// TwinCAT 3 PLC project PLC1
// ProgramVersion: 3.1.4024.0
// libraries:
//   Tc2_ControllerToolbox, * (Beckhoff Automation GmbH)
//   Tc2_MC2, * (Beckhoff Automation GmbH)
//   Tc2_Standard, * (Beckhoff Automation GmbH)
//   Tc2_System, * (Beckhoff Automation GmbH)
//   Tc2_Utilities, * (Beckhoff Automation GmbH)
//   Tc3_Module, * (Beckhoff Automation GmbH)
//   Tc3_Vision, * (Beckhoff Automation GmbH)
// project tree:
//   DUTs/Motion/ E_MotionStates.TcDUT
//   DUTs/Vision/ E_Shapes.TcDUT
//   GVLs/ IO.TcGVL, Motion.TcGVL, Safety.TcGVL
//   / PlcTask.TcTTO
//   POUs/FIle IO/Reading/ FB_ReadReferenceShapeXMLFiles.TcPOU
//   POUs/Indicators/ FB_Flash.TcPOU
//   POUs/ MAIN.TcPOU
//   POUs/Motion/ PositionStateMachine.TcPOU
//   POUs/Vision/ BasicVision.TcPOU
// real-time tasks:
//   TASK PlcTask: cycle T#10ms, priority 20, ADS port 350
//   TASK VnTask ImgAcq (Camera1): cycle T#1ms, priority 5, ADS port 351
//   TASK VnTask ADS (Camera1): cycle T#10ms, priority 6, ADS port 352
// motion (NC):
//   TASK NC-Task 1 SAF: cycle T#2ms, priority 4, ADS port 501
//   TASK NC-Task 1 SVB: cycle T#10ms, priority 8, ADS port 511
//   AXIS Linear Slide (id 3)
//     Dynamic: Acceleration=5485.83, Deceleration=5485.83, Jerk=164575
//     Velo: RefSearch=3.65722, RefSync=3.65722, SlowManual=18.2861, FastManual=109.7166, Fast=365.722, Maximum=365.722
//     OtherSettings: AllowMotionCmdToSlave=true
//     encoder EncType=19
//       EncPara: ScaleFactorNumerator=4.064, ScaleFactorDenominator=1048576, MaxCount=#xffffffff
//         SoftEndMinControl: Range=-5
//         SoftEndMaxControl: Range=275
//     drive DrvType=16
//       DrvPara: MaxCount=#xffffffff, DriveControlDWord=#x00020100
//         Analog: VeloReferenz=402.2942, VeloScale=32, TorqueSetpointScale=10, ScaleFactorActTorque=0.1
//         TimeComp: TaskDelayCycles=1
//     controller CtrType=1
//       CtrPara: PriorControlFactor=1
//         PosDiffControl: Enable=false
//         Observer: BandWidth=20
// I/O:
//   DEVICE EK1100, AmsNetId 169.254.119.130.3.1
//     Term 2 (EK1100) [EK1100 EtherCAT Coupler (2A E-Bus)]
//       Term 3 (EL1012) [EL1012 2Ch. Dig. Input 24V, 10µs]
//       Term 4 (EL1252) [EL1252 2Ch. Fast Dig. Input 24V, 1µs, DC Latch]
//       Term 5 (EL1034) [EL1034 4Ch. Dig. Input 24V, potential-free, 10µs]
//       Term 6 (EL2024) [EL2024 4Ch. Dig. Output 24V, 2A]
//       Term 7 (ELM7222-9016) [ELM7222-9016 2Ch. Servo Terminal (48 V, 8 A RMS, OCT, STO, TwinSAFE Logic)]
//         modules: Module 1 (SAFETY)
//         startup 32785:21 := 0E01 // DRV Motor Settings Ch.1 / Commutation offset
//         startup 32785:27 := 10270000 // DRV Motor Settings Ch.1 / Motor speed limitation
//         startup 28688:11 := FC0D // DRV Outputs Ch.1 / Torque limitation
//         startup 32784:19 := FD00 // DRV Amplifier Settings Ch.1 / Current loop proportional gain
//         startup 32784:18 := 0600 // DRV Amplifier Settings Ch.1 / Current loop integral time
//         startup 32784:21 := 2B000000 // DRV Amplifier Settings Ch.1 / Velocity loop proportional gain
//         startup 32784:20 := 96000000 // DRV Amplifier Settings Ch.1 / Velocity loop integral time
//       Term 8 (EL1904) [EL1904, 4 Ch. Safety Input 24V, TwinSAFE]
//         modules: Module 1 (FSOES)
//       Term 16 (EL2004) [EL2004 4Ch. Dig. Output 24V, 0.5A]
//       Term 17 (EL9011) [EL9011 End Terminal]
//   DEVICE Device 1 (RT-Ethernet Adapter)
// variable links:
//   EK1100 <-> EK1100/Term 2 (EK1100)/Term 7 (ELM7222-9016)
//     Term 2 (EK1100)/Term 8 (EL1904)/Module 1 (FSOES)/TxPDO/FSOE <-> Module 1 (SAFETY)/SAFETY FSoE Connection 1 Receive Message/Message_4
//   EK1100 <-> EK1100/Term 2 (EK1100)/Term 8 (EL1904)
//     Term 2 (EK1100)/Term 7 (ELM7222-9016)/Module 1 (SAFETY)/SAFETY FSoE Connection 1 Send Message/Message_4 <-> Module 1 (FSOES)/RxPDO/FSOE
//   NC-Task 1 SAF/Axes/Linear Slide <-> EK1100/Term 2 (EK1100)/Term 7 (ELM7222-9016)
//     Drive/Inputs/In/nDataIn1 <-> DRV Following error actual value Channel 1/Following error actual value
//     Drive/Inputs/In/nDcOutputTime <-> InfoData/DcOutputShift
//     Drive/Inputs/In/nState1 <-> DRV Statusword Channel 1/Statusword
//     Drive/Inputs/In/nState2 <-> DRV Statusword Channel 1/Statusword @bit 8
//     Drive/Inputs/In/nState4 @bit 1 <-> WcState/InputToggle0
//     Drive/Inputs/In/nState4 <-> WcState/WcState0
//     Drive/Outputs/Out/nCtrl1 <-> DRV Controlword Channel 1/Controlword
//     Drive/Outputs/Out/nCtrl2 <-> DRV Controlword Channel 1/Controlword @bit 8
//     Drive/Outputs/Out/nDataOut1 <-> DRV Target position Channel 1/Target position
//     Enc/Inputs/In/nDataIn1 <-> FB Position Channel 1/Position
//     Enc/Inputs/In/nDcInputTime <-> InfoData/DcInputShift
//     Enc/Inputs/In/nState4 @bit 1 <-> WcState/InputToggle0
//     Enc/Inputs/In/nState4 <-> WcState/WcState0
//   PLC1/PLC1 Instance <-> EK1100/Term 2 (EK1100)/Term 16 (EL2004)
//     PlcTask Outputs/PositionStateMachine.bHandClosed <-> Channel 1/Output
//   PLC1/PLC1 Instance <-> EK1100/Term 2 (EK1100)/Term 3 (EL1012)
//     PlcTask Inputs/IO.bInSafetyRunSwitch <-> Channel 1/Input
//     PlcTask Inputs/PositionStateMachine.bRecalibrate <-> Channel 2/Input
//   PLC1/PLC1 Instance <-> EK1100/Term 2 (EK1100)/Term 4 (EL1252)
//     PlcTask Inputs/IO.bInAckSignal <-> Channel 1/Input
//   PLC1/PLC1 Instance <-> EK1100/Term 2 (EK1100)/Term 5 (EL1034)
//     PlcTask Inputs/PositionStateMachine.bLimitSwitch <-> Channel 1/Input
//   PLC1/PLC1 Instance <-> EK1100/Term 2 (EK1100)/Term 6 (EL2024)
//     PlcTask Outputs/MAIN.bLimitSwitchPower <-> Channel 2/Output
//     PlcTask Outputs/MAIN.bRingLight <-> Channel 1/Output
//   PLC1/PLC1 Instance <-> EK1100/Term 2 (EK1100)/Term 7 (ELM7222-9016)
//     PlcTask Outputs/Safety.bErrorAck <-> Module 1 (SAFETY)/SAFETY Standard Outputdata/Standard In Var 1
//     PlcTask Outputs/Safety.bSafetyRestart <-> Module 1 (SAFETY)/SAFETY Standard Outputdata/Standard In Var 7
//     PlcTask Outputs/Safety.bSafetyRun <-> Module 1 (SAFETY)/SAFETY Standard Outputdata/Standard In Var 2
//   PLC1/PLC1 Instance <-> NC-Task 1 SAF/Axes/Linear Slide
//     PlcTask Inputs/Motion.Servo.NcToPlc <-> Outputs/ToPlc
//     PlcTask Outputs/Motion.Servo.PlcToNc <-> Inputs/FromPlc

CONFIGURATION PLC1
    RESOURCE PLC ON TwinCAT3
        TASK PlcTask(INTERVAL := T#10ms, PRIORITY := 20);
        PROGRAM MAIN WITH PlcTask : MAIN;
    END_RESOURCE
END_CONFIGURATION

// ---- DUTs/Motion/E_MotionStates.TcDUT
//{attribute 'qualified_only'}
{attribute 'strict'}
TYPE E_MotionStates :
(
	// Initialize Motor
	eInitialize := 0,
	
	// Activate Calibration
	eActivateCalibration := 1,
	
	// Calibrate Position
	eCalibrate := 2,
	
	// Scan for shape
	eScanAndGrab := 3,
	
	// Open Hand
	eOpenHand := 4,
	
	// Close Hand
	eCloseHand := 5,
	
	// Position 10 : Start
	eSetTargetPosition_1 := 10,
	eRunToPosition_1 := 11,
	
	// Position 20 : Triangle Box
	eSetTargetPosition_2 := 20,
	eRunToPosition_2 := 21,
	
	// Position 30 : Square Box
	eSetTargetPosition_3 := 30,
	eRunToPosition_3 := 31,
	
	// Position 40 : Circle Box
	eSetTargetPosition_4 := 40,
	eRunToPosition_4 := 41,
	
	// Error Handling
	eErrorState1 := 999
);
END_TYPE

// ---- DUTs/Vision/E_Shapes.TcDUT
//{attribute 'qualified_only'}
{attribute 'strict'}
TYPE E_Shapes :
(
	// No shape
	eNoShape := -1,	

	// Triangle
	eTriangle := 0,
	
	// Circle
	eCircle := 1,
	
	// Square
	eSquare := 2
);
END_TYPE

// ---- GVLs/IO.TcGVL
{attribute 'qualified_only'}
VAR_GLOBAL
	// Acknowledge Error Button | Linked to GPB1
	bInAckSignal AT %I* : BOOL;
	// Safe to run Switch | Linked to GSS1
	bInSafetyRunSwitch AT %I* : BOOL;
	
	// Signal from TwinSAFE Controller | Linked to EStopIndicator Alias
	bInEStopSignal AT %I* : BOOL;
	// Light up indicator | Linked to RPBL1
	bOutEStopIndicator AT %Q* : BOOL;
END_VAR

// ---- GVLs/Motion.TcGVL
{attribute 'qualified_only'}
VAR_GLOBAL
	Servo : AXIS_REF;
END_VAR

// ---- GVLs/Safety.TcGVL
{attribute 'qualified_only'}
VAR_GLOBAL
	// PLC Outputs sent to TwinSAFE Controller
	bErrorAck AT %Q* : BOOL;
	bSafetyRun AT %Q* : BOOL;
	bSafetyRestart AT %Q* : BOOL;
END_VAR

// ---- POUs/MAIN.TcPOU
PROGRAM MAIN
VAR
	// ------------------------------------------- //
	// Outputs
	bLight_GPBL1 AT %Q* 	: 	BOOL;
	bLight_GSSL1 AT %Q* 	: 	BOOL;
	
	// ------------------------------------------- //
	// Motion
	bLimitSwitchPower AT %Q*:	BOOL := TRUE;
	
	// ------------------------------------------- //
	// Indicators
	fbBlink : FB_Flash;
	
	// -------------------------------------------------------------------------------------- //
	// Vision
	bRingLight AT %Q*		:	BOOL := TRUE;
	hr						:	HRESULT;
	fbCamera 				:	FB_VN_GevCameraControl;
	eState 					: 	EtcVNCameraState;
	
	// Raw Input
	ipImageIn 				: 	ITcVnImage;
	
	// ------------------------------------------- //
	// Colors
	
	// Colored output to perform processing on
	ipImageWork 			: 	ITcVnImage;
	ipImageWorkDisp 		: 	ITcVnDisplayableImage;
	
	// Color maps to black and white output
	// ** Could also check for ranges [0,0,0] to [199,255,255] to go straight to proper color map **
	ipImageColorMap_White 	: 	ITcVnImage;
	aColorLow_White 		: 	TcVnVector4_LREAL := [199,255,255];
	aColorHigh_White 		: 	TcVnVector4_LREAL := [255,255,255];
	
	// Invert image so that objects are white and background is black
	ipImageColorMap_Black	: 	ITcVnImage;
	ipImageColorMapDisp_Black : ITcVnDisplayableImage;
	
	// Processed Output
	ipImageResult 			:	ITcVnImage;
	ipImageResultDisp 		: 	ITcVnDisplayableImage;
	
	
	// ------------------------------------------- //
	// Contours
	
	ipContourList 			: 	ITcVnContainer;				// Container of containers containing points for contours
	ipContourListIterator	: 	ITcVnForwardIterator;		// Used to dynamically iterate through ContourList
	ipContour				: 	ITcVnContainer;				// A single contour
	
	aColor_Green			: 	TcVnVector4_LREAL := [0,255,0]; // Constant value, color of drawn contours
	
	// ------------------------------------------- //
	// Object Detection
	
	// Load Reference FIles
	bFilesRead				: 	BOOL := FALSE;
	fbReadReferenceShapeFiles : FB_ReadReferenceShapeXMLFiles;
		
	ipReference_Triangle	: 	ITcVnContainer;				// Destination container for our triangle	
	ipReference_Circle		: 	ITcVnContainer;				// Destination container for our circle
	ipReference_Square		: 	ITcVnContainer;				// Destination container for our square																		
	
	// Calculate area and dissimilarity to determine correct shape type
	fArea					: 	LREAL;						// Area of found contours
	
	fTriangleDissimilarity	: 	LREAL;						// Dissimilarity between reference triangle and actual images
	fCircleDissimilarity	: 	LREAL;						// Dissimilarity between reference circle and actual images
	fSquareDissimilarity	: 	LREAL;						// Dissimilarity between reference square and actual images
	fMinimumDissimilarity	: 	LREAL;						
	
	sText					:	STRING(256);				// Text label on contour
	aCenter					:	TcVnPoint2_LREAL;			// Center of mass of contour
	
	iShape					: 	E_SHAPES := -1;				// Detected shape to be sent to PositionStateMachine
END_VAR

_AppInfo.KeepOutputsOnBP := TRUE;

// Safety Handling
Safety.bSafetyRestart := IO.bInAckSignal;
Safety.bErrorAck := IO.bInAckSignal;
Safety.bSafetyRun := IO.bInSafetyRunSwitch; // ** HARDWIRED TO TRUE **

// Indicators
bLight_GPBL1 := IO.bInAckSignal;
bLight_GSSL1 := IO.bInSafetyRunSwitch;

fbBlink(bEnable:= NOT IO.bInEStopSignal, tTimeOn:= T#500MS, tTimeOff:= T#500MS, bPulse=> IO.bOutEStopIndicator);

// -------------------------------------------------------------------------------------- //
// Vision
	
// Read in reference image files
IF NOT bFilesRead THEN
	fbReadReferenceShapeFiles(
		ipReference_Triangle => ipReference_Triangle,
		ipReference_Circle => ipReference_Circle,
		ipReference_Square => ipReference_Square
	);
	
	bFilesRead := fbReadReferenceShapeFiles.bAllFilesLoaded;
END_IF

IF bFilesRead THEN
	eState := fbCamera.GetState();
	hr := S_OK;
		
	IF eState <= TCVN_CS_ERROR THEN // If state is in error, attempt reset
		hr := fbCamera.Reset();
	ELSIF eState < TCVN_CS_ACQUIRING THEN
		hr := fbCamera.StartAcquisition();
	ELSIF eState = TCVN_CS_ACQUIRING THEN
		// Get current image and set ROI
		hr := fbCamera.GetCurrentImage(ipImageIn);
		//hr := F_VN_SetRoi(953, 480, 450, 370, ipImageIn, hr); 
			
		// Check if image was successfully recieved
		IF SUCCEEDED(hr) AND ipImageIn <> 0 THEN
			// Color Detection
		
			// Create working colored image and displayable version
			hr := F_VN_ConvertColorSpace(ipImageIn, ipImageWork,TCVN_CST_BAYER_RG_TO_RGB, hr);
			hr := F_VN_CopyIntoDisplayableImage(ipImageWork, ipImageWorkDisp, hr);
			
			// Copy our work image into final image for later use during contour drawing
			hr := F_VN_CopyImage(ipImageWork, ipImageResult, hr);
			
			// Increase contrast by converting anything that isn't pure white to black
			// This creates a white image with black shapes on it
			hr := F_VN_CheckColorRange(ipImageWork, ipImageColorMap_White, aColorLow_White, aColorHigh_White, hr);
			
			// Invert white color map to a black color map 
			// This creates a black image with white shapes on it
			hr := F_VN_InvertImageColor(ipImageColorMap_White, ipImageColorMap_Black, hr);
			hr := F_VN_CopyIntoDisplayableImage(ipImageColorMap_Black, ipImageColorMapDisp_Black,hr);
			
			// ------------------------------------------- //
			// Contours
			
			// Use color map to find contours
			hr := F_VN_FindContours(ipImageColorMap_Black, ipContourList,hr);
			
			
			// ** DELETE WHEN ALL REFERENCES CREATED **
			// Count the number of contours and store in iContourSize
			// Write points to XML file
			hr := F_VN_GetForwardIterator(ipContourList, ipContourListIterator, hr);
		
			// Evaluate each subcontainer for contour points
			WHILE SUCCEEDED(hr) AND_THEN ipContourListIterator.CheckIfEnd() <> S_OK DO
				hr := F_VN_GetContainer(ipContourListIterator, ipContour, hr);
				hr := F_VN_IncrementIterator(ipContourListIterator, hr);
				
				// Draw contours
				hr := F_VN_DrawContours(ipContour, -1, ipImageResult, aColor_Green, 3, hr);
				
				// ------------------------------------------- //
				// Shape Detection
				
				// Determine area of contours to save resources scanning miscellaneous junk
				hr := F_VN_ContourArea(ipContour, fArea, hr);
				
				// Compare contours to reference images and determine closest match
				IF fArea > 10000 THEN
					hr := F_VN_MatchContours(ipContour, ipReference_Triangle, TCVN_CMCM_CONTOURS_MATCH_I1, fTriangleDissimilarity, hr);
					
					IF fTriangleDissimilarity < 0.0006 THEN
						iShape := eCircle;
						sText := 'Circle';
					ELSIF fTriangleDissimilarity >= 0.028 AND fTriangleDissimilarity <= 0.033 THEN
						iShape := eSquare;
						sText := 'Square';
					ELSIF fTriangleDissimilarity >= 0.122 AND fTriangleDissimilarity <= 0.144 THEN
						iShape := eTriangle;
						sText := 'Triangle';
					ELSE
						iShape := eNoShape;
						sText := 'Unknown';
					END_IF
				END_IF
				
				// Calculate center of mass and place text onto shape
				hr := F_VN_ContourCenterOfMass(ipContour, aCenter, hr);
				hr := F_VN_PutText(sText, ipImageResult, LREAL_TO_UDINT(aCenter[0] - 60), LREAL_TO_UDINT(aCenter[1] + 10), ETcVnFontType.TCVN_FT_HERSHEY_PLAIN, 2, aColor_Green,hr);
			END_WHILE
			
			hr := F_VN_CopyIntoDisplayableImage(ipImageResult, ipImageResultDisp, hr);
			
		END_IF
	END_IF
	
	// Call to PositionStateMachine to run motion
	PositionStateMachine(iShape := iShape);
END_IF

END_PROGRAM

// ---- POUs/Indicators/FB_Flash.TcPOU
FUNCTION_BLOCK FB_Flash
VAR_INPUT
	bEnable : BOOL;
	tTimeOn : TIME;
	tTimeOff : TIME;
END_VAR
VAR_OUTPUT
	bPulse : BOOL;
END_VAR
VAR
	fbTON : TON; // Timer on delay function block
	fbTOF : TOF; // Timer off delay function block
END_VAR

fbTON(IN := bEnable AND NOT fbTOF.Q, PT := tTimeOff, Q => , ET => );
fbTOF(IN := fbTON.Q, PT := tTimeOn, Q => bPulse, ET => );

END_FUNCTION_BLOCK

// ---- POUs/FIle IO/Reading/FB_ReadReferenceShapeXMLFiles.TcPOU
FUNCTION_BLOCK FB_ReadReferenceShapeXMLFiles

VAR_INPUT
END_VAR

VAR_OUTPUT
	ipReference_Triangle	: 	ITcVnContainer;		// Destination container for our triangle	
	ipReference_Circle		: 	ITcVnContainer;		// Destination container for our circle
	ipReference_Square		: 	ITcVnContainer;		// Destination container for our square
	bAllFilesLoaded			:	BOOL := FALSE;		// Triangle, Circle, and Square files are all loaded
END_VAR

VAR
	fbReadContainer			: 	FB_VN_ReadContainer;// Reads container and compares it to reference
	
	bTriangleReferenceLoaded: 	BOOL := FALSE;		// Triangle file is loaded
	bCircleReferenceLoaded	: 	BOOL := FALSE;		// Circle file is loaded		
	bSquareReferenceLoaded	: 	BOOL := FALSE;		// Square file is loaded

	sTriangleFilePath		: 	STRING(256) := 'C:\Users\Administrator\Documents\Vision\Shapes\ContourTemplates\Original\triangle.xml';		// File path to reference triangle on target system
	sCircleFilePath			: 	STRING(256) := 'C:\Users\Administrator\Documents\Vision\Shapes\ContourTemplates\Original\circle.xml';		// File path to reference circle on target system
	sSquareFilePath			: 	STRING(256) := 'C:\Users\Administrator\Documents\Vision\Shapes\ContourTemplates\Original\rectangle.xml';	// File path to reference square on target system
	
	nTriangleReadId			: 	INT := 0;
	nCircleReadId			: 	INT := 0;
	nSquareReadId			: 	INT := 0;
END_VAR

// Read Triangle
IF NOT bTriangleReferenceLoaded THEN
	fbReadContainer(
		sFilePath:= sTriangleFilePath, 
		ipDestContainer:= ipReference_Triangle, 
		nDestTypeGuid:= , 
		bRead:= TRUE, 
		nTimeout:= T#5S, 
	);
	
	IF NOT fbReadContainer.bBusy THEN
		IF nTriangleReadId >= 2 THEN
			bTriangleReferenceLoaded := TRUE;
		ELSE
			nTriangleReadId := nTriangleReadId + 1;
			fbReadContainer(sFilePath := sTriangleFilePath, bRead := FALSE);
		END_IF
	END_IF
END_IF

// Read Circle
IF NOT bCircleReferenceLoaded THEN
	fbReadContainer(
		sFilePath:= sCircleFilePath, 
		ipDestContainer:= ipReference_Circle, 
		nDestTypeGuid:= , 
		bRead:= TRUE, 
		nTimeout:= T#5S, 
	);
	
	IF NOT fbReadContainer.bBusy THEN
		IF nCircleReadId >= 2 THEN
			bCircleReferenceLoaded := TRUE;
		ELSE
			nCircleReadId := nCircleReadId + 1;
			fbReadContainer(sFilePath := sCircleFilePath, bRead := FALSE);
		END_IF
	END_IF
END_IF

// Read Square
IF NOT bSquareReferenceLoaded THEN
	fbReadContainer(
		sFilePath:= sSquareFilePath, 
		ipDestContainer:= ipReference_Square, 
		nDestTypeGuid:= , 
		bRead:= TRUE, 
		nTimeout:= T#5S, 
	);
	
	IF NOT fbReadContainer.bBusy THEN
		IF nSquareReadId >= 2 THEN
			bSquareReferenceLoaded := TRUE;
		ELSE
			nSquareReadId := nSquareReadId + 1;
			fbReadContainer(sFilePath := sSquareFilePath, bRead := FALSE);
		END_IF
	END_IF
END_IF

IF bTriangleReferenceLoaded AND bSquareReferenceLoaded AND bCircleReferenceLoaded THEN
	bAllFilesLoaded := TRUE;
END_IF

END_FUNCTION_BLOCK

// ---- POUs/Motion/PositionStateMachine.TcPOU
PROGRAM PositionStateMachine
VAR_INPUT
	iShape 					: 	INT;
END_VAR
VAR
	// State Machine
	iMotionStep 			: 	E_MotionStates;
	iNextTargetPosition		:	E_MotionStates;
	iResetState				: 	INT;
	
	// Motion
	iRunSpeed 				: 	INT := 100;
	iTargetPosition			:	INT;
	bExecuteMotion			:	BOOL;
	bRecalibrate AT %I*		:	BOOL;
	iPosition AT %Q* 		: 	LREAL;
	
	fbMotorEnable 			: 	MC_Power;
	fbMoveAbsolute 			: 	MC_MoveAbsolute;
	fbMoveVelocity			:	MC_MoveVelocity;
	fbSetPosition			:	MC_SetPosition;
	fbMotorStop 			: 	MC_Stop;
	fbMotorReset 			: 	MC_Reset;
	fbReadPosition 			: 	MC_ReadActualPosition;
	
	bServoAxisError AT %I* 	: 	BOOL;
	
	bLimitSwitch AT %I*		:	BOOL;
	bHandClosed AT %Q*		:	BOOL;
	
	// Timers
	tHandActuationTimer		:	TON;
	tVisionPauseTimer		:	TON;
	bStartHandTimer			:	BOOL;
	bStartVisionTimer		:	BOOL;
	
	// Vision
	hr						:	HRESULT;
	iNumberOfContours		:	ULINT;
END_VAR

Motion.Servo.ReadStatus();
fbReadPosition(
	Axis:= Motion.Servo, 
	Enable:= TRUE,  
	Position=> iPosition
);

IF bRecalibrate AND NOT fbMoveAbsolute.Busy AND NOT fbMoveVelocity.Busy AND NOT Motion.Servo.Status.Moving AND NOT Motion.Servo.Status.Error THEN
	iMotionStep := eActivateCalibration;
END_IF

	
CASE iMotionStep OF
	
	eInitialize : // Axis Ready
	
		fbMotorEnable(
			Axis:= Motion.Servo, 
			Enable:= TRUE, 
			Enable_Positive:= TRUE, 
			Enable_Negative:= TRUE, 
		);
	
		IF fbMotorEnable.Status THEN
			iMotionStep := eActivateCalibration;
		END_IF
		
	// -------------------------------------------------- //
		
	eActivateCalibration : // Activate Calibration
		bHandClosed := FALSE;
		
		IF bLimitSwitch THEN // Switch is not pressed, calibrate
			fbMoveVelocity(
				Axis:= Motion.Servo, 
				Execute:= TRUE , 
				Velocity:= 20, 
				Direction:= MC_Negative_Direction, 
			);
			iMotionStep := eCalibrate;
		ELSE // Switch is pressed, do not calibrate
			fbMoveVelocity(Axis:= Motion.Servo, Execute:= FALSE);
			fbSetPosition(Axis:= Motion.Servo, Execute:= TRUE, Position:= 0);
			iMotionStep := eSetTargetPosition_1;
		END_IF
		
		IF fbMoveAbsolute.Error THEN
			iMotionStep := eErrorState1;
		END_IF
	
	// -------------------------------------------------- //
	
	eCalibrate : // Axis Calibrating
		fbMoveVelocity(
			Axis:= Motion.Servo, 
			Execute:= FALSE , 
		);
		
		IF NOT bLimitSwitch AND NOT fbMoveVelocity.Busy THEN
			fbSetPosition(Axis:= Motion.Servo, Execute:= TRUE, Position:= 0);
			iMotionStep := eSetTargetPosition_1;
		ELSIF fbMoveVelocity.Error THEN
			iMotionStep := eErrorState1;
		END_IF
	
	// -------------------------------------------------- //
	
	eSetTargetPosition_1 : // Target Position : Start (0mm)
		iTargetPosition := 0;
		bExecuteMotion := TRUE;
		IF fbMoveAbsolute.Busy THEN
			iMotionStep := eRunToPosition_1;
		END_IF
		
		IF fbMoveAbsolute.Error THEN
			iMotionStep := eErrorState1;
		END_IF
	
	// -------------------------------------------------- //
	
	eRunToPosition_1 : // Run to Target Position : Start
		bExecuteMotion := FALSE;
		
		IF fbMoveAbsolute.Done AND NOT fbMoveAbsolute.Busy THEN
			iMotionStep := eScanAndGrab;
		ELSIF fbMoveAbsolute.Error THEN
			iMotionStep := eErrorState1;
		END_IF
	
	// -------------------------------------------------- //
	
	eSetTargetPosition_2 : // Set Target Position : Triangle Box (90mm)
		iTargetPosition := 90;
		bExecuteMotion := TRUE;
		
		iMotionStep := eRunToPosition_2;
		
		IF fbMoveAbsolute.Error THEN
			iMotionStep := eErrorState1;
		END_IF
	
	// -------------------------------------------------- //
	
	eRunToPosition_2 : // Run to Target Position : Triangle Box
		bExecuteMotion := FALSE;
		IF fbMoveAbsolute.Done AND NOT fbMoveAbsolute.Busy THEN
			iMotionStep := eOpenHand;
		ELSIF fbMoveAbsolute.Error THEN
			iMotionStep := eErrorState1;
		END_IF
	
	// -------------------------------------------------- //
	
	eSetTargetPosition_3 : // Set Target Position : Square Box (180mm)
		iTargetPosition := 180;
		bExecuteMotion := TRUE;
		IF fbMoveAbsolute.Busy THEN
			iMotionStep := eRunToPosition_3;
		END_IF
		
		IF fbMoveAbsolute.Error THEN
			iMotionStep := eErrorState1;
		END_IF
	
	// -------------------------------------------------- //
	
	eRunToPosition_3 : // Run to Target Position : Square Box
		bExecuteMotion := FALSE;
		IF fbMoveAbsolute.Done AND NOT fbMoveAbsolute.Busy THEN
			iMotionStep := eOpenHand;
		ELSIF fbMoveAbsolute.Error THEN
			iMotionStep := eErrorState1;
		END_IF
	
	// -------------------------------------------------- //
	
	eSetTargetPosition_4 : // Set Target Position : Circle Box (270mm)
		iTargetPosition := 270;
		bExecuteMotion := TRUE;
		IF fbMoveAbsolute.Busy THEN
			iMotionStep := eRunToPosition_4;
		END_IF
		
		IF fbMoveAbsolute.Error THEN
			iMotionStep := eErrorState1;
		END_IF
	
	// -------------------------------------------------- //
	
	eRunToPosition_4 : // Run to Target Position : Circle Box
		bExecuteMotion := FALSE;
		
		IF fbMoveAbsolute.Done AND NOT fbMoveAbsolute.Busy THEN
			iMotionStep := eOpenHand;
		ELSIF fbMoveAbsolute.Error THEN
			iMotionStep := eErrorState1;
		END_IF
	
	// -------------------------------------------------- //
	
	eScanAndGrab : // Scan for shape and Grab
		hr := F_VN_GetNumberOfElements(Main.ipContourList, iNumberOfContours, hr);
		
		// If some object is present and it's one of our three shapes
		IF iNumberOfContours = 1 AND iShape	<> -1 THEN
			bStartVisionTimer := TRUE;
			// Pause for half a second to allow camera to reliably detect object with no interference
			IF tVisionPauseTimer.Q THEN
				bStartVisionTimer := FALSE;
				CASE iShape OF
					eTriangle :
						iNextTargetPosition := eSetTargetPosition_2;
						iMotionStep := eCloseHand;
					eSquare	:
						iNextTargetPosition := eSetTargetPosition_3;
						iMotionStep := eCloseHand;
					eCircle	:	
						iNextTargetPosition := eSetTargetPosition_4;
						iMotionStep := eCloseHand;
				END_CASE
			END_IF
		END_IF
		
		IF fbMoveAbsolute.Error THEN
			iMotionStep := eErrorState1;
		END_IF
		
	// -------------------------------------------------- //
	
	eOpenHand : // Open hand state before axis information resets
		bHandClosed := FALSE;
		bStartHandTimer := TRUE;
		IF tHandActuationTimer.Q THEN
			bStartHandTimer := FALSE;
			iMotionStep := eSetTargetPosition_1;
		END_IF
		
		IF Motion.Servo.Status.Error THEN
			iMotionStep := eErrorState1;
		END_IF
		
	// -------------------------------------------------- //
	
	eCloseHand : // Close hand state to prevent interference from camera
		bHandClosed := TRUE;
		bStartHandTimer := TRUE;	
		IF tHandActuationTimer.Q THEN
			bStartHandTimer := FALSE;
			iMotionStep := iNextTargetPosition;
		END_IF
		
		IF Motion.Servo.Status.Error THEN
			iMotionStep := eErrorState1;
		END_IF
	
	// -------------------------------------------------- //
	
	eErrorState1 : // Error State 1
		// Disable all motion function blocks
		fbMoveAbsolute(Axis := Motion.Servo, Execute := FALSE);
		fbMoveVelocity(Axis := Motion.Servo, Execute := FALSE);
		// Alternate between enable and disable reset till error clears
		CASE iResetState OF
			0:
				fbMotorEnable(Axis:= Motion.Servo, Enable:= FALSE );
				fbMotorReset(Axis := Motion.Servo, Execute := TRUE);
				iResetState := 1;
			1:
				fbMotorReset(Axis := Motion.Servo, Execute := FALSE);
				iResetState := 0;
		END_CASE
		
		// If reset is successful, move to initialization state
		IF NOT Motion.Servo.Status.Error THEN
			iMotionStep := eInitialize;
		END_IF
	
	// -------------------------------------------------- //
END_CASE

fbMoveAbsolute(
	Axis:= Motion.Servo, 
	Execute:= bExecuteMotion, 
	Position:= iTargetPosition, 
	Velocity:= iRunSpeed, 
);

tHandActuationTimer(IN:= bStartHandTimer, PT:= T#1000MS);
tVisionPauseTimer(IN := bStartVisionTimer, PT := T#500MS);

END_PROGRAM

// ---- POUs/Vision/BasicVision.TcPOU
PROGRAM BasicVision
VAR
		
	hr						:	HRESULT;
	fbCamera 				:	FB_VN_GevCameraControl;
	eState 					: 	EtcVNCameraState;
	
	// Raw Input
	ipImageIn 				: 	ITcVnImage;
	
	// ------------------------------------------- //
	// Colors
	
	// Colored output to perform processing on
	ipImageWork 			: 	ITcVnImage;
	ipImageWorkDisp 		: 	ITcVnDisplayableImage;
	
	// Color maps to black and white output
	ipImageColorMap 		:	ITcVnImage;
	ipImageColorMapDisp 	:	ITcVnDisplayableImage;
	aColorLow_Red 			:	TcVnVector4_LREAL := [0,0,0];				// Red : [50,10,0]
	aColorHigh_Red 			:	TcVnVector4_LREAL := [198,254,254];			// Red : [90,30,15]
	
	// Processed Output
	ipImageResult 			: 	ITcVnImage;
	ipImageResultDisp 		:	ITcVnDisplayableImage;
END_VAR

eState := fbCamera.GetState();
hr := S_OK;

IF eState = TCVN_CS_ERROR THEN // If state is in error, attempt reset
	hr := fbCamera.Reset();
ELSIF eState < TCVN_CS_ACQUIRING THEN
	hr := fbCamera.StartAcquisition();
ELSIF eState = TCVN_CS_ACQUIRING THEN
	hr := fbCamera.GetCurrentImage(ipImageIn);
	
	// Check if image was successfully recieved
	IF SUCCEEDED(hr) AND ipImageIn <> 0 THEN
		// Color Detection
	
		// Create images
		hr := F_VN_ConvertColorSpace(ipImageIn, ipImageWork,TCVN_CST_BAYER_RG_TO_RGB, hr);
		hr := F_VN_CopyIntoDisplayableImage(ipImageWork, ipImageWorkDisp, hr);
		
		// Copy our work image into final image for later use during contour drawing
		// hr := F_VN_CopyImage(ipImageWork, ipImageResult, hr);
	
		// Increase contrast by converting red to white and everything else to black
		hr := F_VN_CheckColorRange(ipImageWork, ipImageColorMap, aColorLow_Red, aColorHigh_Red, hr);
		hr := F_VN_CopyIntoDisplayableImage(ipImageColorMap, ipImageColorMapDisp,hr);
		
		// ------------------------------------------- //
	END_IF
END_IF

END_PROGRAM
